(* PLC project Properties Example.project, CODESYS CODESYS V3.5 SP20 Patch 1 *)
(* stored: creationDateTime 2025-05-23T12:50:11.2423092, modificationDateTime 2025-05-23T12:49:55.2150783 *)

PROGRAM Main
  VAR_INPUT
    MotorA : Motor;
  END_VAR
  VAR
    MotorAIsRunning : BOOL;
  END_VAR

                    
// Set property
MotorA.IsRunning := TRUE;


// Get property
MotorAIsRunning := MotorA.IsRunning;
                  
END_PROGRAM

FUNCTION_BLOCK Motor
  VAR
    _isRunning : BOOL;
  END_VAR

                    
                  

PROPERTY IsRunning : BOOL
GET
                            
// Perform validation if necessary

IsRunning := _isRunning;
                          
END_GET
SET
                            
// Perform validation if necessary

_isRunning := IsRunning;
                          
END_SET
END_PROPERTY
END_FUNCTION_BLOCK

CONFIGURATION Device
  RESOURCE Application ON PLC
    TASK MainTask(INTERVAL := T#20ms, PRIORITY := 1);
    PROGRAM Main WITH MainTask : Main;
  END_RESOURCE
END_CONFIGURATION
